PROGRAM BarcodeCtrl_Utac
VAR
	bTestsensor:BOOL;
	(*X120_00*)

END_VAR

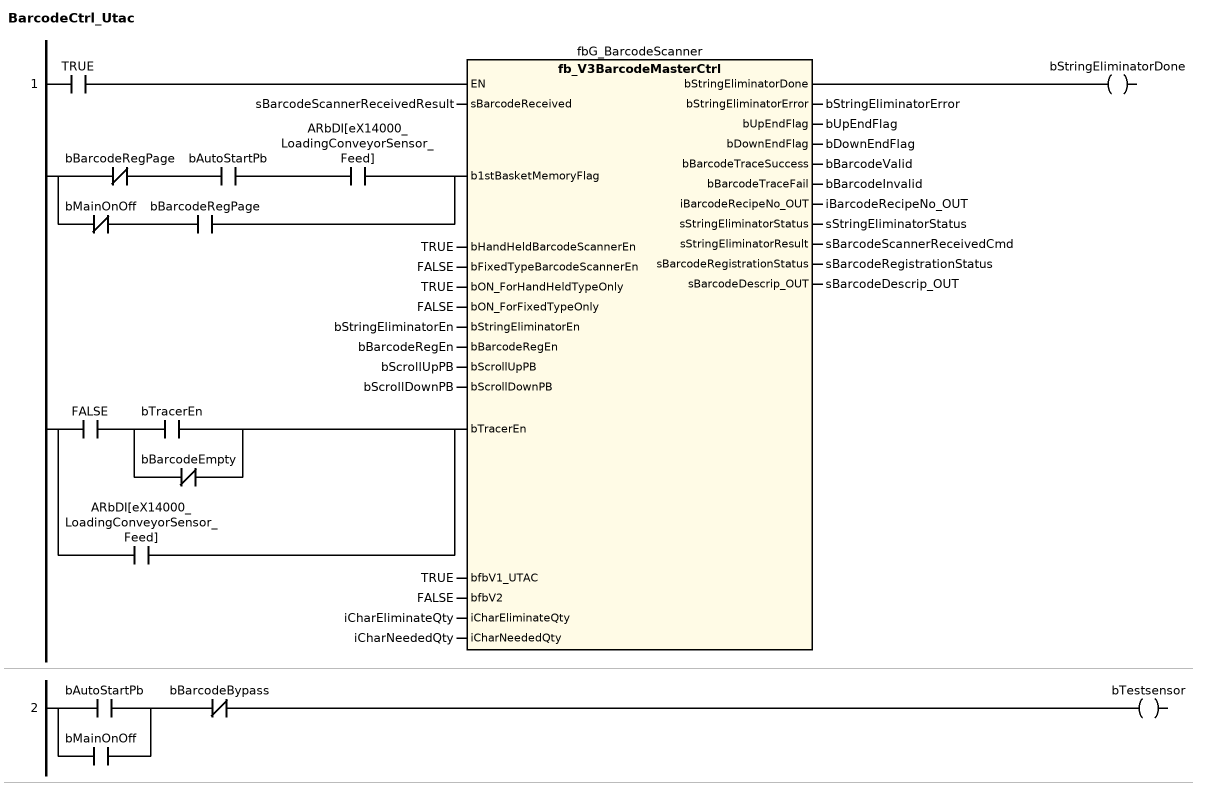
// NETWORK 1
fbG_BarcodeScanner(
    sBarcodeReceived := sBarcodeScannerReceivedResult,
    b1stBasketMemoryFlag := NOT bBarcodeRegPage AND bAutoStartPb AND ARbDI[eX14000_LoadingConveyorSensor_Feed] OR NOT bMainOnOff AND bBarcodeRegPage,
    bHandHeldBarcodeScannerEn := TRUE,
    bFixedTypeBarcodeScannerEn := FALSE,
    bON_ForHandHeldTypeOnly := TRUE,
    bON_ForFixedTypeOnly := FALSE,
    bStringEliminatorEn := bStringEliminatorEn,
    bBarcodeRegEn := bBarcodeRegEn,
    bScrollUpPB := bScrollUpPB,
    bScrollDownPB := bScrollDownPB,
    bTracerEn := FALSE AND (bTracerEn OR NOT bBarcodeEmpty) OR ARbDI[eX14000_LoadingConveyorSensor_Feed],
    bfbV1_UTAC := TRUE,
    bfbV2 := FALSE,
    iCharEliminateQty := iCharEliminateQty,
    iCharNeededQty := iCharNeededQty,
    bStringEliminatorError => bStringEliminatorError,
    bUpEndFlag => bUpEndFlag,
    bDownEndFlag => bDownEndFlag,
    bBarcodeTraceSuccess => bBarcodeValid,
    bBarcodeTraceFail => bBarcodeInvalid,
    iBarcodeRecipeNo_OUT => iBarcodeRecipeNo_OUT,
    sStringEliminatorStatus => sStringEliminatorStatus,
    sStringEliminatorResult => sBarcodeScannerReceivedCmd,
    sBarcodeRegistrationStatus => sBarcodeRegistrationStatus,
    sBarcodeDescrip_OUT => sBarcodeDescrip_OUT); // fb_V3BarcodeMasterCtrl
bStringEliminatorDone := fbG_BarcodeScanner.bStringEliminatorDone;

// NETWORK 2
bTestsensor := (bAutoStartPb OR bMainOnOff) AND NOT bBarcodeBypass;

END_PROGRAM

(* stored: Version 1.1.0.1, ProductVersion 3.1.4024.12
   POU BarcodeCtrl_Utac: Id {a6729c8d-a0c6-46ee-950f-e7a3277999df}, SpecialFunc None *)
